TYPE ST_ParamRecipe :
STRUCT
	
END_STRUCT
END_TYPE

(* stored: Version 1.1.0.1, ProductVersion 3.1.4020.6
   DUT ST_ParamRecipe: Id {39f85e54-6d8b-42f2-ae8f-3e8767f14653} *)
